FUNCTION_BLOCK Q_ActiveMask (* Command change active mask( Part 6 - F.34 ) *)
  (* Standard: ISO 11783-6; Description: Copyright (c) 2022 HR Agrartechnik GmbH This program and the accompanying materials are made available under the terms of the Eclipse Public License 2.0 which is available at https://www.eclipse.org/legal/epl-2.0/ SPDX-License-Identifier: EPL-2.0 see Description Tab *)
  (* Version 1.0, 2022-07-08, Franz Höpfinger, HR Agrartechnik GmbH *)
  PACKAGE isobus::UT::Q;
  IMPORT isobus::UT::Q::const::IDs::ID_NULL;
  (* Documentation:
  Command change active mask( Part 6 - F.34 )
   This command is used to change the active mask of a working set to either a data or an alarm mask object.
   Note: The WorkingSet Object ID (u16WorkSetId) is fixed to 0 by the authors of logiBUS®. The user must ensure that the WorkingSet object in the object pool always has Object ID 0. This is the default in most tools (e.g., ISO-Designer by Bucher Automation AG, or Isobus Studio by to-the-future / Tobias Tenberg). Since there is only one WorkingSet object, this restriction does not cause any practical limitation.
   Valid Object IDs
   A new-active-mask Object ID is valid if it falls within one of the following ISO 11783-6 ID ranges (Annex F.34):
    - DataMask: 1000 – 1999
   - AlarmMask: 2000 – 2999
    ID_NULL (65535) is not a valid command target for the new active mask. Any ID outside these ranges is invalid for commanding.
   param[in] {u16NewMaskId, uint16_t}
   Object ID of new active (data/alarm)-mask
   Return Values (s16result):
   int16_t
    - VT_E_NO_ERR (0) - OK
   - VT_E_NOT_READY (-131) - VT client not yet ready
   - VT_E_OVERFLOW (-6) - buffer overflow
   - VT_E_NOACT (-8) - Command not possible in current state
   - VT_E_NO_INSTANCE (-21) - No VT client available
   - VT_E_ISO_INSTANCE_INVALID (-129) - Identifier for instance (connection) invalid
   - VT_E_NOT_ALIVE (-130) - Identifier for instance valid, but VT Dead.
   - VT_OK_BUFFERED (18) - command buffered, waiting for VT to be ready
  *)
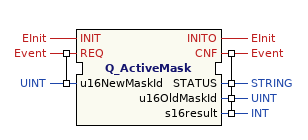
  EVENT_INPUT
    INIT : EInit; (* Service Initialization *)
    REQ WITH u16NewMaskId; (* Service Request *)
  END_EVENT
  EVENT_OUTPUT
    INITO : EInit; (* Initialization Confirm *)
    CNF WITH STATUS, u16OldMaskId, s16result, u16OldMaskId; (* Confirmation of Requested Service *)
  END_EVENT
  VAR_INPUT
    u16NewMaskId : UINT := ID_NULL; (* Object ID of new active (data/alarm)-mask *)
  END_VAR
  VAR_OUTPUT
    STATUS : STRING; (* Service Status *)
    u16OldMaskId : UINT; (* Object ID of old active (data/alarm)-mask *)
    s16result : INT; (* retval see description *)
  END_VAR
END_FUNCTION_BLOCK
